Staubli VAL3: clkValve8.pgx

program clkValve8()
begin
  call toggleValve(8)
end
